FUNCTION Convert_DT_TO_SINT : Hresult
VAR_INPUT
	in : DT;
	out : REFERENCE TO SINT;
END_VAR
VAR
	converted : SINT;
END_VAR

converted := DT_TO_SINT(in);

IF (SINT_TO_DT(converted) <> in) THEN
	Convert_DT_TO_SINT := INCOMPATIBLE;
	RETURN;
END_IF

out := converted;

END_FUNCTION

(* stored: Version 1.1.0.1, ProductVersion 3.1.4024.12
   POU Convert_DT_TO_SINT: Id {203e5a88-2862-44f3-a9cb-70c4e94ef66d}, SpecialFunc None *)
